% RSLogix 500 project P1_KOBIERSKI_M.RSS, saved by version 8.30.00.16 %
PROJECT "UNTITLED"    % processor: Bul.1763 MicroLogix 1100 Series B %

PROGRAM FILES
  LAD 2 "MAIN"  3 rungs
  LAD 3 "IO"  5 rungs
  LAD 4 "CTRL"  7 rungs

DATA FILES
  O0 OUTPUT  4 elements
  I1 INPUT  6 elements
  S2 STATUS  66 elements
  B3 BINARY  1 elements
  T4 TIMER  4 elements
  C5 COUNTER  1 elements
  R6 CONTROL  1 elements
  N7 INTEGER  1 elements
  F8 FLOAT  1 elements

LADDER 2 "MAIN"
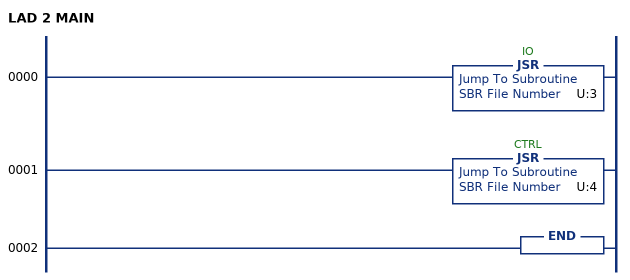
% Rung: 0 %
SOR JSR U:3 EOR
%   U:3  "IO" %
% Rung: 1 %
SOR JSR U:4 EOR
%   U:4  "CTRL" %
% Rung: 2 %
SOR END EOR

LADDER 3 "IO"
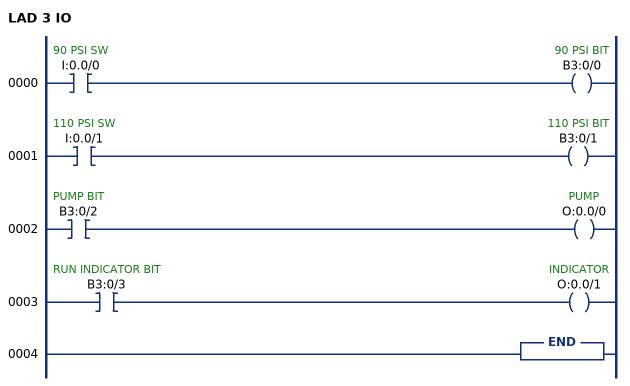
% Rung: 0 %
SOR XIC I:0.0/0 OTE B3:0/0 EOR
%   I:0.0/0  "90 PSI SW" %
%   B3:0/0  "90 PSI BIT" %
% Rung: 1 %
SOR XIC I:0.0/1 OTE B3:0/1 EOR
%   I:0.0/1  "110 PSI SW" %
%   B3:0/1  "110 PSI BIT" %
% Rung: 2 %
SOR XIC B3:0/2 OTE O:0.0/0 EOR
%   B3:0/2  "PUMP BIT" %
%   O:0.0/0  "PUMP" %
% Rung: 3 %
SOR XIC B3:0/3 OTE O:0.0/1 EOR
%   B3:0/3  "RUN INDICATOR BIT" %
%   O:0.0/1  "INDICATOR" %
% Rung: 4 %
SOR END EOR

LADDER 4 "CTRL"
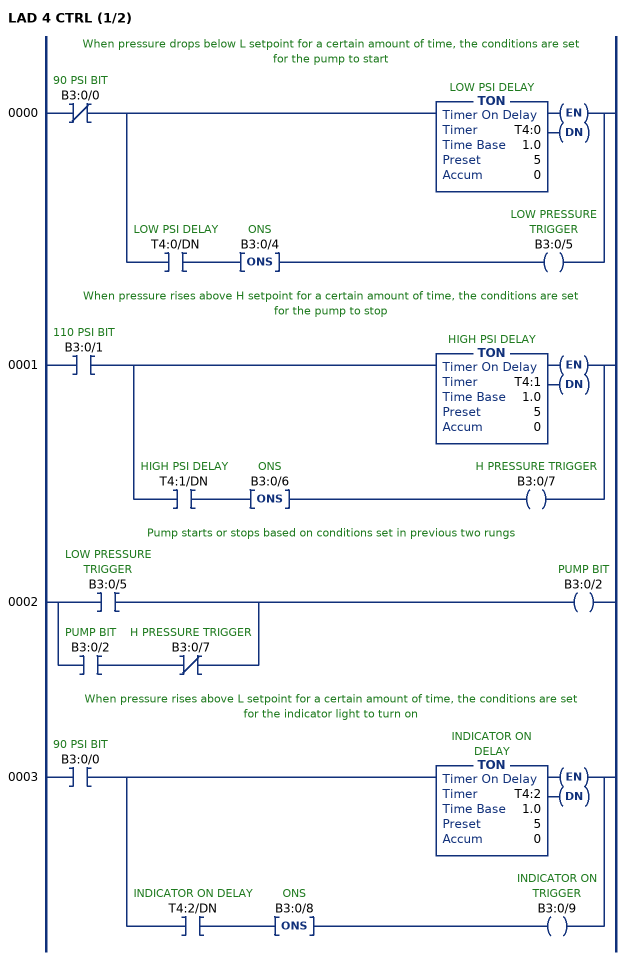
% Rung: 0 %
% When pressure drops below L setpoint for a certain amount of time, the conditions are set for the pump to start %
SOR XIO B3:0/0 BST TON T4:0 1.0 5 0 NXB XIC T4:0/DN ONS B3:0/4 OTE B3:0/5 BND EOR
%   B3:0/0  "90 PSI BIT" %
%   T4:0  "LOW PSI DELAY" %
%   B3:0/4  "ONS" %
%   B3:0/5  "LOW PRESSURE TRIGGER" %
% Rung: 1 %
% When pressure rises above H setpoint for a certain amount of time, the conditions are set for the pump to stop %
SOR XIC B3:0/1 BST TON T4:1 1.0 5 0 NXB XIC T4:1/DN ONS B3:0/6 OTE B3:0/7 BND EOR
%   B3:0/1  "110 PSI BIT" %
%   T4:1  "HIGH PSI DELAY" %
%   B3:0/6  "ONS" %
%   B3:0/7  "H PRESSURE TRIGGER" %
% Rung: 2 %
% Pump starts or stops based on conditions set in previous two rungs %
SOR BST XIC B3:0/5 NXB XIC B3:0/2 XIO B3:0/7 BND OTE B3:0/2 EOR
%   B3:0/5  "LOW PRESSURE TRIGGER" %
%   B3:0/2  "PUMP BIT" %
%   B3:0/7  "H PRESSURE TRIGGER" %
% Rung: 3 %
% When pressure rises above L setpoint for a certain amount of time, the conditions are set for the indicator light to turn on %
SOR XIC B3:0/0 BST TON T4:2 1.0 5 0 NXB XIC T4:2/DN ONS B3:0/8 OTE B3:0/9 BND EOR
%   B3:0/0  "90 PSI BIT" %
%   T4:2  "INDICATOR ON DELAY" %
%   B3:0/8  "ONS" %
%   B3:0/9  "INDICATOR ON TRIGGER" %

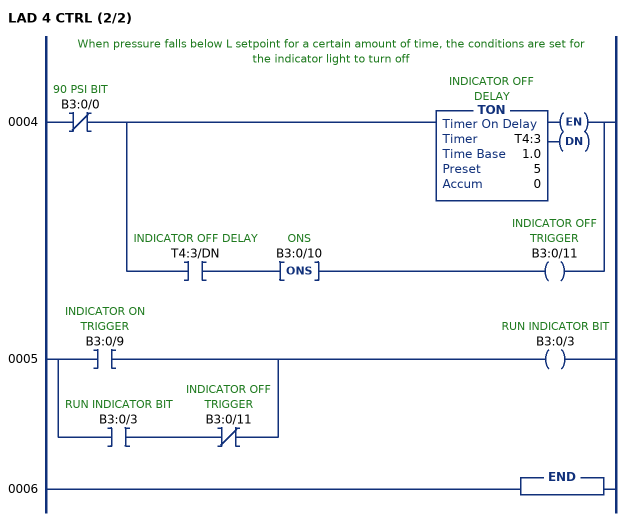
% Rung: 4 %
% When pressure falls below L setpoint for a certain amount of time, the conditions are set for the indicator light to turn off %
SOR XIO B3:0/0 BST TON T4:3 1.0 5 0 NXB XIC T4:3/DN ONS B3:0/10 OTE B3:0/11 BND EOR
%   B3:0/0  "90 PSI BIT" %
%   T4:3  "INDICATOR OFF DELAY" %
%   B3:0/10  "ONS" %
%   B3:0/11  "INDICATOR OFF TRIGGER" %
% Rung: 5 %
SOR BST XIC B3:0/9 NXB XIC B3:0/3 XIO B3:0/11 BND OTE B3:0/3 EOR
%   B3:0/9  "INDICATOR ON TRIGGER" %
%   B3:0/3  "RUN INDICATOR BIT" %
%   B3:0/11  "INDICATOR OFF TRIGGER" %
% Rung: 6 %
SOR END EOR

COMMENTS NOT ATTACHED TO A CURRENT RUNG
  T4:0: When pressure stays below L for a period of time, condition is set to turn pump on

REVISION NOTES
  0: Better naming, added timer

DATA TABLE (non-zero values as saved)
DATA T4
% .PRE .ACC %
% T4:0 % 5 0
% T4:1 % 5 0
% T4:2 % 5 0
% T4:3 % 5 0
